PROGRAM ControlSystem
VAR
		// Variables
	emergencyTime   : TIME := T#10S;
	resetLatch : BOOL := FALSE;
	stateAlarm : AlarmState;
	
		// Function Blocks
	initializer : FB_defaultValues;
END_VAR

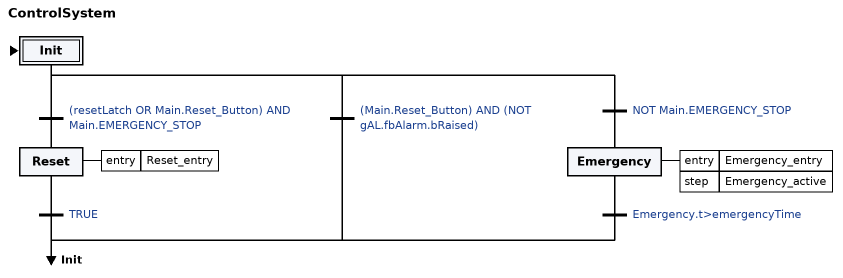
INITIAL_STEP Init:
END_STEP
TRANSITION FROM Init TO Reset
    := (resetLatch OR Main.Reset_Button) AND Main.EMERGENCY_STOP;
END_TRANSITION
STEP Reset:
    Reset_entry(P1);  // entry action
END_STEP
TRANSITION FROM Reset TO Init
    := TRUE;
END_TRANSITION
TRANSITION FROM Init TO Init
    := (Main.Reset_Button) AND (NOT gAL.fbAlarm.bRaised);
END_TRANSITION
TRANSITION FROM Init TO Emergency
    := NOT Main.EMERGENCY_STOP;
END_TRANSITION
STEP Emergency:
    Emergency_entry(P1);  // entry action
    Emergency_active(N);  // step action
END_STEP
TRANSITION FROM Emergency TO Init
    := Emergency.t>emergencyTime;
END_TRANSITION

ACTION Emergency_active:

IF ( (Main.EMERGENCY_STOP) AND (NOT Main.Reset_Button) ) THEN
	resetLatch := TRUE;
	stateAlarm := AlarmState.AlarmClearPreTimer;
END_IF
END_ACTION

ACTION Emergency_entry:

gAL.Motor_ON_OFF := FALSE;				// Stop Motor
gAL.Flow_Valve_1_Percentage  := 100;	// Open all valves
gAL.Level_Valve_1_Percentage := 100;
gAL.Level_Valve_2_Percentage := 100;
gAL.Level_Valve_3_Percentage := 100;

stateAlarm := AlarmState.AlarmActive;
END_ACTION

ACTION Reset_entry:

initializer(MotorState  := gAL.Motor_ON_OFF,
			MotorSpeed  := gAL.Motor_speed_Percentage,
			FV1_Percent := gAL.Flow_Valve_1_Percentage,
			LV1_Percent := gAL.Level_Valve_1_Percentage,
			LV2_Percent := gAL.Level_Valve_2_Percentage,
			LV3_Percent := gAL.Level_Valve_3_Percentage);
			
stateAlarm := AlarmState.AlarmCleared;
END_ACTION

END_PROGRAM

(* stored: Version 1.1.0.1, ProductVersion 3.1.4024.12
   POU ControlSystem: Id {8d9995cd-0e03-49a0-80ce-f3b4149aa1e8}, SpecialFunc None
   Action Emergency_active: Id {f3d9c642-3825-4f1f-8f2e-6190e18b09ed}
   Action Emergency_entry: Id {8fa4c7b6-7e3d-4cd7-9142-9712b4ff052c}
   Action Reset_entry: Id {daed5b0f-1655-4d32-9d05-3f98606b998b} *)
